TYPE ST_GC_SVID :
STRUCT
	SingleProcess : ST_GCSingleProcessStatus;
END_STRUCT
END_TYPE

(* stored: Version 1.1.0.1, ProductVersion 3.1.4026.18
   DUT ST_GC_SVID: Id {98e4cb40-6ac8-4b71-a899-4a314197da67} *)
